(* IEC 61131-3 sources: POMIRTS_lab3/AS/Library/LoopConR/V1.17.0, 3 files *)

(* ---- LoopConR.typ ---- *)
(********************************************************************
 * COPYRIGHT (C) BERNECKER + RAINER, AUSTRIA, A-5142 EGGELSBERG
 ********************************************************************
 * Library: LoopConR
 * File: LoopConR.typ
 * Created: 11.11.2003
 ********************************************************************
 * Global data types of library LoopConR
 ********************************************************************)
TYPE
	lcrCurveByPoints_TabEntry_type : STRUCT
		x	: REAL ;
		y	: REAL ;
	END_STRUCT;
	lcrpid_addPar_typ : STRUCT
		y_autotune_on	: REAL ;
		y_autotune_off	: REAL ;
		t_autotune_max	: REAL ;
		diff_dx_max	: INT ;
		diff_dt_max	: UDINT ;
		osc_nrPeriods	: UINT ;
		optSwitches	: UINT ;
		dY_max	: REAL ;
		Tf_Tv	: REAL ;
		Kw	: REAL ;
		Kfbk	: REAL ;
		fbk_mode	: USINT ;
		d_mode	: USINT ;
		calc_mode	: USINT ;
	END_STRUCT;
	lcrpid_internal_typ : STRUCT
		size	: UINT ;
		valid	: BOOL ;
		autotune_addpar	: lcrpid_addPar_typ ;
		WX_max	: REAL ;
		WX_min	: REAL ;
		invert	: BOOL ;
		deadband	: REAL ;
		dY_max	: REAL ;
		Kp	: REAL ;
		Kp_Tn	: REAL ;
		Tv_Tf	: REAL ;
		Tf_reciproc	: REAL ;
		Kw	: REAL ;
		Kfbk_Kp	: REAL ;
		fbk_mode	: USINT ;
		d_mode	: USINT ;
		force_mode	: USINT ;
		Y_force	: REAL ;
		W	: REAL ;
		X	: REAL ;
		pid_init	: USINT ;
		Yp1	: DINT ;
		Yp2	: DINT ;
		dYi1	: DINT ;
		dYi2	: DINT ;
		Yi1	: DINT ;
		Yi2	: DINT ;
		dt_Tf	: REAL ;
		a11	: DINT ;
		a12	: DINT ;
		a21	: DINT ;
		a22	: DINT ;
		Yd1	: DINT ;
		Yd2	: DINT ;
		Ytotal1	: DINT ;
		Ytotal2	: DINT ;
		Ylim1	: DINT ;
		Ylim2	: DINT ;
		Y1	: DINT ;
		Y2	: DINT ;
		e_fbk	: REAL ;
	END_STRUCT;
END_TYPE

(* ---- LoopConR.fun ---- *)
(********************************************************************
 * COPYRIGHT (C) BERNECKER + RAINER, AUSTRIA, A-5142 EGGELSBERG
 ********************************************************************
 * Library: LoopConR
 * File: LoopConR.fun
 * Created: 11.11.2003
 ********************************************************************
 * Functions and function blocks of library LoopConR
 ********************************************************************)
FUNCTION_BLOCK LCRTimeBasedOnOff
	VAR_INPUT
		enable	:BOOL;
		x	:REAL;
		max_value	:REAL;
		min_value	:REAL;
		timpulse	:REAL;
		tchange_up	:REAL;
		tchange_down	:REAL;
		ref	:BOOL;
	END_VAR
	VAR_OUTPUT
		status	:UINT;
		up	:BOOL;
		down	:BOOL;
		hysteresis_up	:REAL;
		hysteresis_down	:REAL;
		refOk	:BOOL;
	END_VAR
	VAR
		counter_state	:UINT;
		bootkey_old	:UDINT;
		systicks_old	:UDINT;
		musecs_old	:UINT;
		ref_old	:BOOL;
		t_cnt_1	:DINT;
		t_cnt_2	:DINT;
		y_dbl_1	:DINT;
		y_dbl_2	:DINT;
		sysInfo_inst	:SysInfo;
	END_VAR
END_FUNCTION_BLOCK
FUNCTION_BLOCK LCRPWM
	VAR_INPUT
		enable	:BOOL;
		x	:REAL;
		max_value	:REAL;
		min_value	:REAL;
		t_min_pulse	:REAL;
		t_period	:REAL;
	END_VAR
	VAR_OUTPUT
		status	:UINT;
		pulse	:BOOL;
		t_on	:REAL;
		t_off	:REAL;
	END_VAR
	VAR
		counter_state	:UINT;
		bootkey_old	:UDINT;
		systicks_old	:UDINT;
		musecs_old	:UINT;
		cnt_terron_1	:DINT;
		cnt_terron_2	:DINT;
		cnt_terroff_1	:DINT;
		cnt_terroff_2	:DINT;
		cnt_t_pulse_1	:DINT;
		cnt_t_pulse_2	:DINT;
		sysinfo_inst	:SysInfo;
	END_VAR
END_FUNCTION_BLOCK
FUNCTION_BLOCK LCRMovAvgFlt
	VAR_INPUT
		enable	:BOOL;
		x	:REAL;
		base	:UINT;
	END_VAR
	VAR_OUTPUT
		status	:UINT;
		y	:REAL;
	END_VAR
	VAR
		sum_old_dbl_1	:DINT;
		sum_old_dbl_2	:DINT;
		x_old	:ARRAY[0..31] OF REAL;
		p_xold	:UDINT;
		i_xold	:UINT;
		base_old	:UINT;
		enable_old	:BOOL;
		bootkey_old	:UDINT;
	END_VAR
END_FUNCTION_BLOCK
FUNCTION_BLOCK LCRLimScal
	VAR_INPUT
		x	:REAL;
		x1	:REAL;
		y1	:REAL;
		x2	:REAL;
		y2	:REAL;
	END_VAR
	VAR_OUTPUT
		y	:REAL;
	END_VAR
END_FUNCTION_BLOCK
FUNCTION_BLOCK LCRLimit
	VAR_INPUT
		in	:REAL;
		max_value	:DINT;
		min_value	:DINT;
	END_VAR
	VAR_OUTPUT
		status	:UINT;
		out	:DINT;
		max_limit	:BOOL;
		min_limit	:BOOL;
	END_VAR
END_FUNCTION_BLOCK
FUNCTION_BLOCK LCRIntegrate
	VAR_INPUT
		enable	:BOOL;
		x	:REAL;
		tn	:REAL;
		y_max	:REAL;
		y_min	:REAL;
		y_set	:REAL;
		set	:BOOL;
	END_VAR
	VAR_OUTPUT
		status	:UINT;
		y	:REAL;
		max_limit	:BOOL;
		min_limit	:BOOL;
	END_VAR
	VAR
		counter_state	:UINT;
		bootkey_old	:UDINT;
		systicks_old	:UDINT;
		musecs_old	:UINT;
		y_dbl_1	:DINT;
		y_dbl_2	:DINT;
		sysinfo_inst	:SysInfo;
	END_VAR
END_FUNCTION_BLOCK
FUNCTION_BLOCK LCRRamp
	VAR_INPUT
		enable	:BOOL;
		x	:REAL;
		dy_up	:REAL;
		dy_down	:REAL;
		y_max	:REAL;
		y_min	:REAL;
		y_set	:REAL;
		set	:BOOL;
	END_VAR
	VAR_OUTPUT
		status	:UINT;
		y	:REAL;
		x_reached	:BOOL;
		max_limit	:BOOL;
		min_limit	:BOOL;
	END_VAR
	VAR
		counter_state	:UINT;
		bootkey_old	:UDINT;
		systicks_old	:UDINT;
		musecs_old	:UINT;
		y_dbl_1	:DINT;
		y_dbl_2	:DINT;
		sysinfo_inst	:SysInfo;
	END_VAR
END_FUNCTION_BLOCK
FUNCTION_BLOCK LCRPT1
	VAR_INPUT
		enable	:BOOL;
		x	:REAL;
		t	:REAL;
		y_set	:REAL;
		set	:BOOL;
	END_VAR
	VAR_OUTPUT
		status	:UINT;
		y	:REAL;
	END_VAR
	VAR
		counter_state	:UINT;
		bootkey_old	:UDINT;
		systicks_old	:UDINT;
		musecs_old	:UINT;
		y_dbl_1	:DINT;
		y_dbl_2	:DINT;
		sysinfo_inst	:SysInfo;
	END_VAR
END_FUNCTION_BLOCK
FUNCTION_BLOCK LCRContinServo
	VAR_INPUT
		enable	:BOOL;
		x	:REAL;
		max_value	:REAL;
		min_value	:REAL;
		t_impulse	:REAL;
		t_change_up	:REAL;
		t_change_down	:REAL;
		ref	:BOOL;
	END_VAR
	VAR_OUTPUT
		status	:UINT;
		up	:BOOL;
		down	:BOOL;
		hysteresis_up	:REAL;
		hysteresis_down	:REAL;
		refOk	:BOOL;
	END_VAR
	VAR
		counter_state	:UINT;
		bootkey_old	:UDINT;
		systicks_old	:UDINT;
		musecs_old	:UINT;
		ref_old	:BOOL;
		t_cnt_1	:DINT;
		t_cnt_2	:DINT;
		y_dbl_1	:DINT;
		y_dbl_2	:DINT;
		sysInfo_inst	:SysInfo;
	END_VAR
END_FUNCTION_BLOCK
FUNCTION_BLOCK LCRPIDpara
	VAR_INPUT
		enable	:BOOL;
		enter	:BOOL;
		WX_max	:REAL;
		WX_min	:REAL;
		invert	:BOOL;
		deadband	:REAL;
		dY_max	:REAL;
		Kp	:REAL;
		Tn	:REAL;
		Tv	:REAL;
		Tf	:REAL;
		Kw	:REAL;
		Kfbk	:REAL;
		fbk_mode	:USINT;
		d_mode	:USINT;
	END_VAR
	VAR_OUTPUT
		status	:UINT;
		ident	:UDINT;
	END_VAR
	VAR
		internal_data	:lcrpid_internal_typ;
	END_VAR
END_FUNCTION_BLOCK
FUNCTION_BLOCK LCRCurveByPoints
	VAR_INPUT
		x	:REAL;
		NoOfPoints	:UINT;
		ptr_table	:REFERENCE TO lcrCurveByPoints_TabEntry_type;
	END_VAR
	VAR_OUTPUT
		status	:UINT;
		y	:REAL;
	END_VAR
	VAR
		i_tab	:INT;
		iterations	:UINT;
		scal1	:LCRScal;
	END_VAR
END_FUNCTION_BLOCK
FUNCTION_BLOCK LCRScal
	VAR_INPUT
		x	:REAL;
		x1	:REAL;
		y1	:REAL;
		x2	:REAL;
		y2	:REAL;
	END_VAR
	VAR_OUTPUT
		y	:REAL;
	END_VAR
END_FUNCTION_BLOCK
FUNCTION_BLOCK LCRPID
	VAR_INPUT
		enable	:BOOL;
		ident	:UDINT;
		W	:REAL;
		X	:REAL;
		Y_max	:REAL;
		Y_min	:REAL;
		A	:REAL;
		Y_man	:REAL;
		Y_fbk	:REAL;
		hold_I	:BOOL;
		mode	:USINT;
	END_VAR
	VAR_OUTPUT
		status	:UINT;
		e	:REAL;
		Y	:REAL;
		Yp	:REAL;
		Yi	:REAL;
		Yd	:REAL;
	END_VAR
	VAR
		counter_state	:UINT;
		bootkey_old	:UDINT;
		systicks_old	:UDINT;
		musecs_old	:UINT;
		Tv_Tf_old	:REAL;
		enable_old	:BOOL;
		e_old	:REAL;
		deadband_state	:UINT;
		sysinfo_inst	:SysInfo;
		scal_inst	:LCRScal;
	END_VAR
END_FUNCTION_BLOCK

(* ---- LoopConR.var ---- *)
(********************************************************************
 * COPYRIGHT (C) BERNECKER + RAINER, AUSTRIA, A-5142 EGGELSBERG
 ********************************************************************
 * Library: LoopConR
 * File: LoopConR.var
 * Created: 11.11.2003
 ********************************************************************
 * Constants of library LoopConR
 ********************************************************************)
VAR CONSTANT
	LCR_ERR_LCRContinServo_TIMPULSE	: UINT	:= 12036;
	LCR_ERR_LCRCurveByPoints_TABLE	: UINT	:= 12045;
	LCR_ERR_LCRContinServo_TCHANGE	: UINT	:= 12035;
	LCR_ERR_LCRPID_PAR_WX_MAXMIN	: UINT	:= 12043;
	LCR_ERR_LCRRamp_DYUP_DYDOWN	: UINT	:= 12034;
	LCR_ERR_LCRPID_PAR_DEADBAND	: UINT	:= 12044;
	LCRPID_MODE_FREEZE_JOLTFREE	: USINT	:= 105;
	LCR_WARN_LCRPID_YMAN_LIMIT	: UINT	:= 12009;
	LCR_WARN_LCRPID_YFBK_LIMIT	: UINT	:= 12003;
	LCR_WARN_LCRPID_I_MINLIMIT	: UINT	:= 12002;
	LCR_WARN_LCRPID_I_MAXLIMIT	: UINT	:= 12001;
	LCR_ERR_LCRPID_PAR_FBKMODE	: UINT	:= 12024;
	LCRPID_MODE_CLOSE_JOLTFREE	: USINT	:= 104;
	LCR_ERR_LCRMovAvgFlt_BASE	: UINT	:= 12017;
	LCRPID_MODE_OPEN_JOLTFREE	: USINT	:= 103;
	LCR_ERR_LCRPWM_TMINPULSE	: UINT	:= 12032;
	LCR_ERR_LCRPID_PAR_DYMAX	: UINT	:= 12023;
	LCR_ERR_LCRPID_PAR_DMODE	: UINT	:= 12022;
	LCRPID_MODE_MAN_JOLTFREE	: USINT	:= 102;
	LCR_WARN_LCRPID_A_LIMIT	: UINT	:= 12008;
	LCR_ERR_LCRPID_PAR_KFBK	: UINT	:= 12025;
	LCR_ERR_LCRIntegrate_TN	: UINT	:= 12016;
	LCR_ERR_LCRPWM_TPERIOD	: UINT	:= 12033;
	LCR_ERR_LCRPID_PARADAT	: UINT	:= 12020;
	LCRPID_FBK_MODE_INTERN	: USINT	:= 1;
	LCRPID_FBK_MODE_EXTERN	: USINT	:= 2;
	LCR_ERR_LCRPID_PAR_TV	: UINT	:= 12030;
	LCR_ERR_LCRPID_PAR_TN	: UINT	:= 12029;
	LCR_ERR_LCRPID_PAR_TF	: UINT	:= 12028;
	LCR_ERR_LCRPID_PAR_KW	: UINT	:= 12027;
	LCR_ERR_LCRPID_PAR_KP	: UINT	:= 12026;
	LCR_ERR_LCRPID_IDENT	: UINT	:= 12018;
	LCR_ERR_LCRPID_MODE	: UINT	:= 12019;
	LCRPID_MODE_FREEZE	: USINT	:= 5;
	LCRPID_MODE_CLOSE	: USINT	:= 4;
	LCR_ERR_LCRPT1_T	: UINT	:= 12031;
	LCR_ERR_DISABLED	: UINT	:= 65534;
	LCRPID_MODE_OPEN	: USINT	:= 3;
	LCRPID_MODE_AUTO	: USINT	:= 1;
	LCRPID_MODE_MAN	: USINT	:= 2;
	LCRPID_D_MODE_X	: USINT	:= 1;
	LCRPID_D_MODE_E	: USINT	:= 2;
	LCR_WARN_Tx_DT	: UINT	:= 12007;
	LCR_ERR_MAXMIN	: UINT	:= 12037;
	LCR_ERROR	: UINT	:= 12015;
END_VAR
